Universal Robots PolyScope program: _adminCG-WXYZLoadMillMakeLid.urp

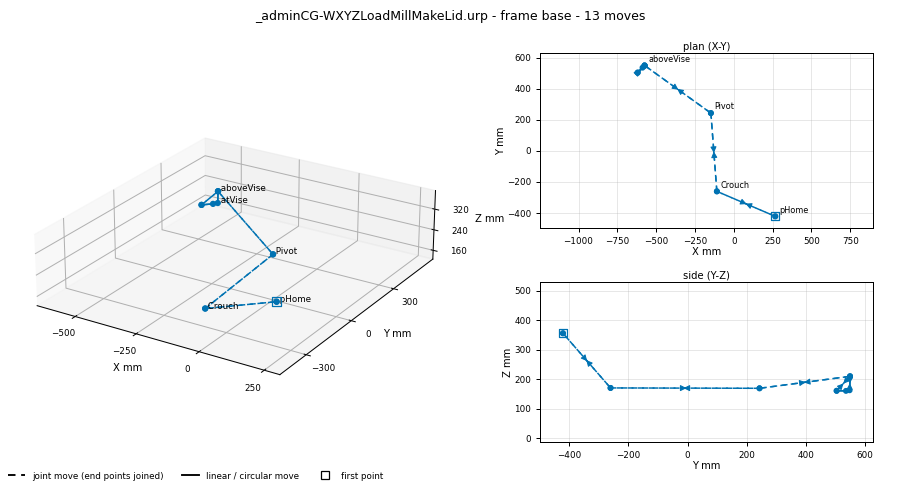
[picture p0: tool path of _adminCG-WXYZLoadMillMakeLid.urp in frame base, 13 of 13 moves have a stored position in this frame; points joined in program order, loops and branches not executed]
Program _adminCG-WXYZLoadMillMakeLid (installation=admin directory=/programs/WED_9AM createdIn=3.8.0.61336 lastSavedIn=3.15.8.106339 robotSerialNumber=2015350924)
Calibrated DH parameters: a=[0, -0.425, -0.39225, 0, 0, 0]; d=[0.089159, 0, 0, 0.10915, 0.09465, 0.0823]; alpha=[1.570796, 0, 0, 1.570796, -1.570796, 0]; deltaTheta=[0, 0, 0, 0, 0, 0]
BeforeStart
  Script file /programs/R2CScript.script
    | # Copyright 2020 VersaBuilt, Inc. All Rights Reserved
    | 
    | global vbR2CIPAddr = "192.168.2.1"
    | global vbR2CPort = 9002
    | global vbVersaBlast = "VERSABLAST"
    | global vbGripperOpen = "GRIPPER_OPEN"
    | global vbGripperClose = "GRIPPER_CLOSE"
    | global vbVise1Open = "VISE_1_OPEN"
    | global vbVise1Close = "VISE_1_CLOSE"
    | global vbVise1Sensor = "VISE_1_SENSOR"
    | global vbVise2Open = "VISE_2_OPEN"
    | global vbVise2Close = "VISE_2_CLOSE"
    | global vbVise2Sensor = "VISE_2_SENSOR"
    | global vbDoorOpen = "DOOR_OPEN"
    | global vbDoorOpenSensor = "DOOR_OPEN_SENSOR"
    | global vbDoorOpenSensor2 = "DOUBLE_DOOR_OPEN_SENSOR"
    | global vbDoorClose = "DOOR_CLOSE"
    | global vbDoorCloseSensor = "DOOR_CLOSE_SENSOR"
    | global vbDoorCloseSensor2 = "DOUBLE_DOOR_CLOSE_SENSOR"
    | global vbDoor = "SingleDoor"
    | global vbDoorWaitTime = 7
    | global vbDoorTimeOut = 15
    | global vbDoorSensors = True
    | global vbViseSensors = True
    | global vbSim = False
    | 
    | def InitializeR2CVars():
    |   vbR2CIPAddr = vbSaveR2CIPAddr
    |   vbDoor = vbSaveDoor
    |   vbDoorSensors = vbSaveDoorSensors
    |   vbViseSensors = vbSaveViseSensors
    |   vbDoorWaitTime = vbSaveDoorWaitTime
    | end
    | 
    | def SetIPAddr(ip):
    |   vbSaveR2CIPAddr = ip
    | end
    | 
    | # Send a R2C Command. If the response is an error, a blocking popup will be generated.
    | # Otherwise the response is returned
    | def SendR2CCommand(text):
    |   response = SendR2CCommandRaw(text)
    |   CheckR2CResponse(response)
    |   return response
    | end
    | 
    | # Reads a R2C response and creates a blocking popup if an error is detected
    | def CheckR2CResponse(response):
    |   errorPortion = str_sub(response, 0, 5)
    |   if (errorPortion == "ERROR"):
    |     popup("Robot2CNC Error, press the Stop Program button and resolve the error condition: " + response, error = True, blocking = True)
    |     halt
    |   end
    | end
    | 
    | def OpenSocket():
    |   count = 0
    |   socket_result = socket_open(vbR2CIPAddr, vbR2CPort, "socket_1")
    |   while (not(socket_result) and count < 10):
    |     sleep(1)
    |     count = count + 1
    |     socket_result = socket_open(vbR2CIPAddr, vbR2CPort, "socket_1")
    |   end
    |   if not(socket_result):
    |     popup("Communication with Robot2CNC Failed (socket open). Press the Stop Program button and fix the Robot2CNC communication problem.", "Robot2CNC Command Error", error = True, blocking = True)
    |     halt
    |   end
    | end
    | 
    | # Send a R2C command, return the response. Does not check response for error.
    | def SendR2CCommandRaw(text):
    |   InitializeR2CVars()
    |   count = 0
    |   while count < 3:
    |     count = count + 1
    |     OpenSocket()
    |     socket_send_line(text, "socket_1")
    |     status = socket_read_string("socket_1", "", ";", True, 5)
    |     socket_close("socket_1")
    |     if str_len(status) > 0:
    |       return status
    |     end
    |     sleep(1)
    |   end
    |   popup("Communication with Robot2CNC Failed (no response). Press the Stop Program button and fix the Robot2CNC communication problem.", "Robot2CNC Command Error", error = True, blocking = True)
    |   halt
    | end
    | 
    | def VersaBlastOn():
    |     if vbSim == False:
    |         SetDO(vbVersaBlast, "ON")
    |     end
    | end
    | 
    | def VersaBlastOff():
    |     if vbSim == False:
    |         SetDO(vbVersaBlast, "OFF")
    |     end
    | end
    | 
    | def OpenGripper():
    |     if vbSim == False:
    |         SetDO(vbGripperClose, "OFF")
    |         SetDO(vbGripperOpen, "ON")
    |     end
    | end
    | 
    | def CloseGripper():
    |     if vbSim == False:
    |         SetDO(vbGripperClose, "ON")
    |         SetDO(vbGripperOpen, "OFF")
    |     end
    | end
    | 
    | def FloatGripper():
    |     if vbSim == False:
    |         SetDO(vbGripperClose, "OFF")
    |         SetDO(vbGripperOpen, "OFF")
    |     end
    | end
    | 
    | def OpenVise(viseNum):
    |   if vbSim == False:
    |     if viseNum == 1 :
    |       SetDO(vbVise1Close, "OFF")
    |       SetDO(vbVise1Open, "ON")
    |     else:
    |       SetDO(vbVise2Close, "OFF")
    |       SetDO(vbVise2Open, "ON")
    |     end
    |   end
    | end
    | 
    | def CloseVise(viseNum):
    |   if vbSim == False:
    |     if viseNum == 1 :
    |       SetDO(vbVise1Open, "OFF")
    |       SetDO(vbVise1Close, "ON")
    |     else:
    |       SetDO(vbVise2Open, "OFF")
    |       SetDO(vbVise2Close, "ON")
    |     end
    |   end
    | end
    | 
    | def ViseFumbleCheck(viseNum):
    |   if vbSim == False:
    |     InitializeR2CVars()
    |     if vbViseSensors:
    |       if viseNum == 1:
    |         if (GetDI(vbVise1Sensor) == "OFF"):
    |           popup("Vise fumble. The VB Mill App Kit could not confirm the part was loaded in the vise. Exiting","VB Mill App Kit",error= True, blocking=True)
    |           halt
    |         end
    |       else:
    |         if (GetDI(vbVise2Sensor) == "OFF"):
    |           popup("Vise fumble. The VB Mill App Kit could not confirm the part was loaded in the vise. Exiting","VB Mill App Kit",error= True, blocking=True)
    |           halt
    |         end
    |       end
    |     end
    |   end
    | end
    | 
    | # clamps a vise by moving in the direction specified by ODID
    | def ClampVise(viseNum,ODID):
    |   if vbSim == False:
    |     if (ODID == "OD"):
    |       CloseVise(viseNum)
    |     else:
    |       OpenVise(viseNum)
    |     end
    |   end
    | end
    | 
    | def UnClampVise(viseNum,ODID):
    |   if vbSim == False:
    |     if (ODID == "OD"):
    |       OpenVise(viseNum)
    |     else:
    |       CloseVise(viseNum)
    |     end
    |   end
    | end
    | 
    | def OpenDoor():
    |   if vbSim == False:
    |     InitializeR2CVars()
    |     if vbDoor != "CNCDoor" :
    |       SetDO(vbDoorClose, "OFF")
    |       SetDO(vbDoorOpen, "ON")
    |       if vbDoorSensors == True :
    |         vbDoorTimeOutCounter = 0
    |         while GetDI(vbDoorOpenSensor) == "OFF" :
    |           sleep(.1)
    |           vbDoorTimeOutCounter = vbDoorTimeOutCounter + 0.1
    |           if vbDoorTimeOutCounter >= vbDoorTimeOut :
    |             FloatDoor()
    |             popup("Door failed to open within " + to_str(vbDoorTimeOut) + " seconds (door sensor 1).<br><br>Fix the problem, open the door and press Continue or press the Stop button.", blocking = True)
    |             vbDoorTimeOutCounter = 0
    |           end
    |         end
    |         # if we have double doors, check the double door sensor
    |         if (vbDoor == "DoubleDoor") :
    |           vbDoorTimeOutCounter = 0
    |           while GetDI(vbDoorOpenSensor2) == "OFF" :
    |             sleep(.1)
    |             vbDoorTimeOutCounter = vbDoorTimeOutCounter + 0.1
    |             if vbDoorTimeOutCounter >= vbDoorTimeOut :
    |               FloatDoor()
    |               popup("Door failed to open within " + to_str(vbDoorTimeOut) + " seconds (door sensor 2).<br><br>Fix the problem, open the door and press Continue or press the Stop button.", blocking = True)
    |               vbDoorTimeOutCounter = 0
    |             end
    |           end
    |         end
    |       else:
    |         sleep(vbDoorWaitTime)
    |       end
    |       # give it another second to open all the way...
    |       sleep(1)
    |       # Float the door after open/close
    |       FloatDoor()
    |     else:
    |       sleep(vbDoorWaitTime)
    |     end
    |   end
    | end
    | 
    | def CloseDoor():
    |   if vbSim == False:
    |     InitializeR2CVars()
    |     if vbDoor != "CNCDoor" :
    |       SetDO(vbDoorOpen, "OFF")
    |       SetDO(vbDoorClose, "ON")
    |       if vbDoorSensors == True :
    |         vbDoorTimeOutCounter = 0
    |         while GetDI(vbDoorCloseSensor) == "OFF" :
    |           sleep(.1)
    |           vbDoorTimeOutCounter = vbDoorTimeOutCounter + 0.1
    |           if vbDoorTimeOutCounter >= vbDoorTimeOut :
    |             FloatDoor()
    |             popup("Door failed to close within " + to_str(vbDoorTimeOut) + " seconds (door sensor 1).<br><br>Fix the problem, open the door and press Continue or press the Stop button.", blocking = True)
    |             vbDoorTimeOutCounter = 0
    |           end
    |         end
    |         # if we have double doors, check the double door sensor
    |         if (vbDoor == "DoubleDoor") :
    |           vbDoorTimeOutCounter = 0
    |           while GetDI(vbDoorCloseSensor2) == "OFF" :
    |             sleep(.1)
    |             vbDoorTimeOutCounter = vbDoorTimeOutCounter + 0.1
    |             if vbDoorTimeOutCounter >= vbDoorTimeOut :
    |               FloatDoor()
    |               popup("Door failed to close within " + to_str(vbDoorTimeOut) + " seconds (door sensor 2).<br><br>Fix the problem, open the door and press Continue or press the Stop button.", blocking = True)
    |               vbDoorTimeOutCounter = 0
    |             end
    |           end
    |         end
    |       else:
    |         sleep(vbDoorWaitTime)
    |       end
    |       # give it another second to close tight...
    |       sleep(1)
    |       # Float door after closing/opening
    |       FloatDoor()
    |     else:
    |       sleep(vbDoorWaitTime)
    |     end
    |   end
    | end
    | 
    | # Wait for DI at addr to equal value, timeout after specified seconds. Retuens true on success, false on timeout.
    | def WaitDI(addr, value, timeout):
    |   if vbSim == False:
    |     time = 0
    |     while GetDI(addr) != value:
    |       sleep(.1)
    |       time = time + 0.1
    |       if time > timeout:
    |         return False
    |       end
    |     end
    |     return True
    |   else:
    |     return True
    |   end
    | end
    | 
    | def SetDO(ioAddress, onOff):
    |   if vbSim == False:
    |     command = "SET_DO," + ioAddress + "," + onOff + ";"
    |     result = SendR2CCommand(command)
    |     if result + ";" != command:
    |       popup("Error setting digital output on Robot2CNC, press Stop Program and resolve error.<br>Unable to set " + to_str(ioAddress) + ", " + to_str(onOff), error=True, blocking = True)
    |       halt
    |     end
    |   end
    | end
    | 
    | def GetDI(ioAddress):
    |   if vbSim == False:
    |     command = "GET_DI," + ioAddress + ";"
    |     result = SendR2CCommand(command)
    |     return str_sub(result, str_len(command))
    |   end
    | end
    | 
    | def WaitCNC():
    |   if vbSim == False:
    |     status = SendR2CCommand("CNC_STATUS;")
    |     while (status != "CNC_STATUS,COMPLETE"):
    |       status = SendR2CCommand("CNC_STATUS;")
    |       sleep(0.5)
    |     end
    |     if (status != "CNC_STATUS,COMPLETE"):
    |       popup("Can not Validate Program Completion<br>CNC Status: " + status, "Milling Program Not Complete", False, False, blocking = True)
    |       halt
    |     else:
    |       SendR2CCommand("RESET_CNC;")
    |     end
    |   end
    | end
    | 
    | def FloatVise(viseNum):
    |   if vbSim == False:
    |     if viseNum == 1 :
    |       SetDO(vbVise1Open, "OFF")
    |       SetDO(vbVise1Close, "OFF")
    |     else:
    |       SetDO(vbVise2Open, "OFF")
    |       SetDO(vbVise2Close, "OFF")
    |     end
    |   end
    | end
    | 
    | def FloatDoor():
    |   if vbSim == False:
    |     SetDO(vbDoorOpen, "OFF")
    |     SetDO(vbDoorClose, "OFF")
    |   end
    | end
    | 
    | def RunCNCProgram(progNum):
    |   if vbSim == False:
    |     status = SendR2CCommand("CNC_STATUS;")
    |     if not(status == "CNC_STATUS,IDLE" or status == "CNC_STATUS,COMPLETE"):
    |       popup("CNC Not Idle. Press Stop Program and resolve problem on CNC.<br>Result from CNC: " + status, "CNC Not Ready", False, False, blocking = True)
    |       halt
    |     end
    |     SendR2CCommand("RUN_PROGRAM,"+to_str(progNum)+";")
    |   end
    | end
    | 
    | def SetHaasCellSafe():
    |   if vbSim == False:
    |     SendR2CCommand("ENABLE_HAAS_CELL_SAFE;")
    |   end
    |   sleep(0.1)
    | end
    | 
    | def ClearHaasCellSafe():
    |   if vbSim == False:
    |     SendR2CCommand("DISABLE_HAAS_CELL_SAFE;")
    |   end
    | end
    | 
    | def GetMacro(macroNum):
    |   if vbSim == False :
    |     send = "READ_MACRO,"+to_str(macroNum)
    |     length = str_len(send)
    |     result = SendR2CCommand(send+";")
    |     return to_num(str_sub(result,length+1))
    |   else:
    |     return 0
    |   end
    | end
    | 
    | def SetMacro(macroNum, value):
    |   if vbSim == False:
    |     result = SendR2CCommand("WRITE_MACRO,"+to_str(macroNum)+","+to_str(value)+";")
    |   end
    | end
Robot Program (runOnlyOnce=true)
  URCap Robot2CNC (VersaBuilt Robot2CNC, VersaBuilt Robotics Inc.) dataModel(text1=100, getFunction=Run CNC Program)
  URCap Robot2CNC (VersaBuilt Robot2CNC, VersaBuilt Robotics Inc.) dataModel(getFunction=Wait for CNC Program)
  Set DigitalOutput pin=digital_out[1]; digitalValue=0
  MoveJ speed 180 deg/s, acceleration 120 deg/s^2 (useActiveTCP=true)
    Waypoint pHome: TCP in base x=267.143 y=-421.455 z=355.857 mm, rx=1.114 ry=1.106 rz=0.0051 rad; joints [-44.997, -90.001, -89.999, -90.001, 90.004, 0.008] deg; flange x=267.141 y=-421.459 z=431.857 mm, rx=-1.2021 ry=2.9025 rz=0.0001 rad
  Call _adminLinearIndex4
  MoveJ speed 180 deg/s, acceleration 80 deg/s^2 (useActiveTCP=true)
    Waypoint Crouch: motionParameters(blendRadius=0.1); TCP in base x=-109.147 y=-260.51 z=170.949 mm, rx=1.6765 ry=0.1344 rz=-1.0823 rad; joints [-90.001, -61.532, -138.324, -70.319, 90.003, 35.526] deg; flange x=-109.151 y=-260.743 z=246.949 mm, rx=-0.9582 ry=-2.991 rz=-0.0046 rad
    Waypoint Pivot: TCP in base x=-147.635 y=243.514 z=169.706 mm, rx=1.5686 ry=-1.56 rz=-2.2133 rad; joints [-216.207, -62.031, -138.326, -69.682, 89.953, 8.126] deg; flange x=-147.713 y=243.495 z=245.705 mm, rx=2.8953 ry=1.219 rz=0.0016 rad
    Waypoint aboveVise: TCP in base x=-574.214 y=549.766 z=210.179 mm, rx=1.5691 ry=-1.5593 rz=-2.2096 rad; joints [-215.874, -135.166, -47.777, -87.171, 90.057, 8.324] deg; flange x=-574.293 y=549.916 z=286.179 mm, rx=2.8919 ry=1.2217 rz=0.0003 rad
  MoveL speed 250 mm/s, acceleration 1200 mm/s^2 (useActiveTCP=true) feature=Base
    Waypoint atVise: TCP in base x=-574.631 y=548.367 z=163.046 mm, rx=1.569 ry=-1.559 rz=-2.2097 rad; joints [-215.773, -135.921, -53.364, -80.82, 90.054, 8.421] deg; flange x=-574.703 y=548.506 z=239.046 mm, rx=2.892 ry=1.2218 rz=0.0002 rad
    Set DigitalOutput pin=digital_out[0]; digitalValue=0
    Wait Sleep waitTime=1
    Waypoint aboveVise: TCP in base x=-574.214 y=549.766 z=210.179 mm, rx=1.5691 ry=-1.5593 rz=-2.2096 rad; joints [-215.874, -135.166, -47.777, -87.171, 90.057, 8.324] deg; flange x=-574.293 y=549.916 z=286.179 mm, rx=2.8919 ry=1.2217 rz=0.0003 rad
    Set DigitalOutput pin=digital_out[0]; digitalValue=1
    Wait Sleep waitTime=1
  MoveJ speed 60 deg/s, acceleration 80 deg/s^2 (useActiveTCP=true)
    Waypoint besideVise: TCP in base x=-618.827 y=504.439 z=161.279 mm, rx=1.5691 ry=-1.5594 rz=-2.2095 rad; joints [-211.341, -136.66, -52.299, -81.153, 90.067, 12.859] deg; flange x=-618.907 y=504.592 z=237.279 mm, rx=2.8919 ry=1.2216 rz=0.0003 rad
  MoveL speed 50 mm/s, acceleration 20 mm/s^2 (useActiveTCP=true) feature=Base
    Waypoint pushBlock: TCP in base x=-587.818 y=535.971 z=161.001 mm, rx=1.569 ry=-1.5592 rz=-2.2097 rad; joints [-214.484, -136.176, -53.211, -80.718, 90.059, 9.715] deg; flange x=-587.889 y=536.114 z=237.001 mm, rx=2.892 ry=1.2217 rz=0.0002 rad
    Set DigitalOutput pin=digital_out[1]; digitalValue=1
    Wait Sleep waitTime=1
    Waypoint besideVise: TCP in base x=-618.827 y=504.439 z=161.279 mm, rx=1.5691 ry=-1.5594 rz=-2.2095 rad; joints [-211.341, -136.66, -52.299, -81.153, 90.067, 12.859] deg; flange x=-618.907 y=504.592 z=237.279 mm, rx=2.8919 ry=1.2216 rz=0.0003 rad
  MoveJ speed 60 deg/s, acceleration 80 deg/s^2 (useActiveTCP=true)
    Waypoint aboveVise: TCP in base x=-574.214 y=549.766 z=210.179 mm, rx=1.5691 ry=-1.5593 rz=-2.2096 rad; joints [-215.874, -135.166, -47.777, -87.171, 90.057, 8.324] deg; flange x=-574.293 y=549.916 z=286.179 mm, rx=2.8919 ry=1.2217 rz=0.0003 rad
  MoveJ speed 60 deg/s, acceleration 80 deg/s^2 (useActiveTCP=true)
    Waypoint Pivot: TCP in base x=-147.635 y=243.514 z=169.706 mm, rx=1.5686 ry=-1.56 rz=-2.2133 rad; joints [-216.207, -62.031, -138.326, -69.682, 89.953, 8.126] deg; flange x=-147.713 y=243.495 z=245.705 mm, rx=2.8953 ry=1.219 rz=0.0016 rad
    Waypoint Crouch: motionParameters(blendRadius=0.1); TCP in base x=-109.147 y=-260.51 z=170.949 mm, rx=1.6765 ry=0.1344 rz=-1.0823 rad; joints [-90.001, -61.532, -138.324, -70.319, 90.003, 35.526] deg; flange x=-109.151 y=-260.743 z=246.949 mm, rx=-0.9582 ry=-2.991 rz=-0.0046 rad
    Waypoint pHome: TCP in base x=267.143 y=-421.455 z=355.857 mm, rx=1.114 ry=1.106 rz=0.0051 rad; joints [-44.997, -90.001, -89.999, -90.001, 90.004, 0.008] deg; flange x=267.141 y=-421.459 z=431.857 mm, rx=-1.2021 ry=2.9025 rz=0.0001 rad
    Set DigitalOutput pin=digital_out[0]; digitalValue=0
  URCap Robot2CNC (VersaBuilt Robot2CNC, VersaBuilt Robotics Inc.) dataModel(getFunction=Run CNC Program, text1=332)
SubProgram  [hidden by the author, left out]
SubProgram _adminLinearIndex4 [hidden by the author, left out]
